{attribute 'qualified_only'}
VAR_GLOBAL
	start_button : BOOL;
	stop_button : BOOL;
	auto_button : BOOL;
	manual_button : BOOL;
	joy_x : LREAL;
	joy_y : LREAL;
	joy_button : BOOL;
END_VAR

(* stored: Version 1.1.0.1, ProductVersion 3.1.4024.12
   GVL visual_box_GVL: Id {89c43190-6e1b-499a-9ff7-91a688e80191} *)
